FUNCTION F_RadToDeg : LREAL
VAR_INPUT
	fRad :LREAL;
END_VAR
VAR
END_VAR

F_RadToDeg := fRad * (180/PI);

END_FUNCTION

(* stored: Version 1.1.0.1, ProductVersion 3.1.4024.10
   POU F_RadToDeg: Id {f37597c2-ea64-4fce-8450-e12d5fb83a5c}, SpecialFunc None *)
